TEXTLIST TL_FbStateTimer
  0 = 'UNDEFINED'
  1 = 'RUN'
  2 = 'STOP'
  3 = 'SAFE'
  8 = 'DELAY OUT'
  9 = 'DELAY IN'
   = ''
END_TEXTLIST

(* stored: Version 1.1.0.1, ProductVersion 3.1.4022.12
   TextList TL_FbStateTimer: Id {6bfdda5b-1ec1-437c-9fe2-ebfed0f2e196} *)
